Staubli VAL3: loadProcessList.pgx

public program loadProcessList(num& x_nResult[])
// load the process list
  local num i
  local string l_sMessage
  local string l_sMessage2
begin
  // setMutex
  setMutex(cycleStatus:bMutex)
  // load a different processList
  if cycleStatus:bCycle==false and cycleStatus:bSimulation==false
    //saveData:sPathPList+x_sProcess
    x_nResult=saveCycle:libLoad(saveData:sPathPList)
    delay(0)
    if saveData:bDebug and x_nResult!=0
      logMsg("[KERNEL] SETPROCESSLIST:Loading processList, CODE: "+toString("",x_nResult))
    endIf
    // check the result
    if x_nResult!=0
      // load the template and empty the list
      x_nResult=saveCycle:libLoad("kernel/template/session/saveCycle")
      delay(0)
      libDelete(saveData:sPathPList)
      saveCycle:libSave(saveData:sPathPList)
      // default process list has been charged
      call language:message(l_sMessage,-7)
      call language:message(l_sMessage2,97)
      popUpMsg(l_sMessage+"saveCycle... "+l_sMessage2)
    endIf
  else
    x_nResult=-1
  endIf
  //release
  cycleStatus:bMutex=false
end
